INTERFACE I_TOD EXTENDS I_Datatype

PROPERTY PUBLIC Value : REFERENCE TO TOD
GET
END_GET
END_PROPERTY

END_INTERFACE

(* stored: Version 1.1.0.1, ProductVersion 3.1.4024.15
   Itf I_TOD: Id {1287ebd8-bfc7-08d3-1630-07183c36c7ff}
   Property Value: Id {322e0b2e-9721-03ce-0c48-76d61b637e0e}
   Get Get: Id {1edb240b-9c84-0e68-1b77-4871ed6973b9} *)
